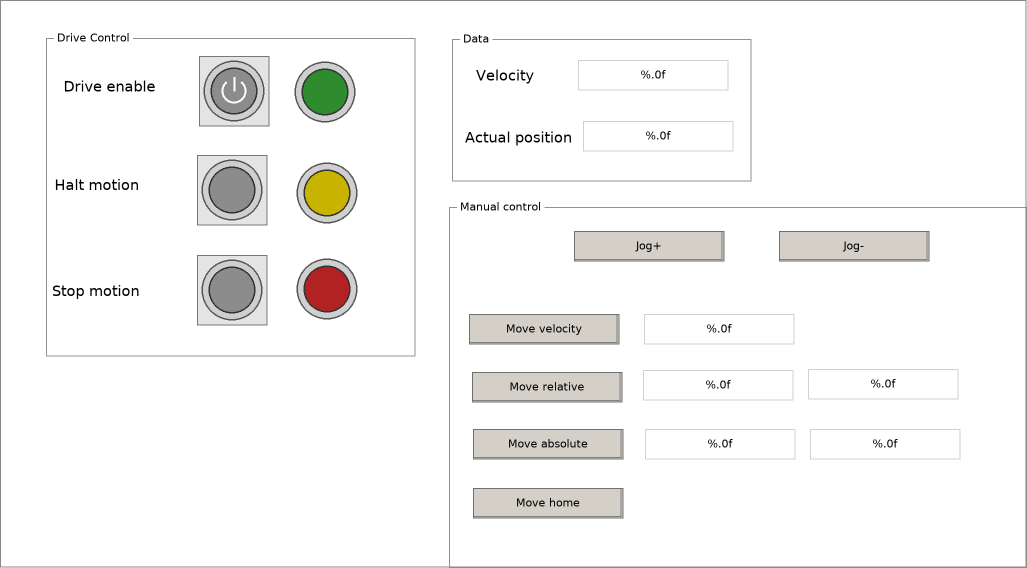
VISUALIZATION HMI  // 1027x568
    GroupBox (46,30 369x326), "Drive Control"
        PowerSwitch (153,26 70x70), variable: MAIN.AxisControl.McPowerEnable, behaviour: TOGGLE, style: Switch-PowerSwitch-Gray
        Lamp1 (244,27 70x70), variable: MAIN.AxisControl.AxisStatus, style: Lamp-Lamp1-Green
        PushSwitch (151,125 70x70), variable: MAIN.AxisControl.ExecuteHalt, behaviour: TOGGLE, style: Switch-PushSwitch-Gray
        PushSwitch (151,225 70x70), variable: MAIN.AxisControl.ExecuteStop, behaviour: TOGGLE, style: Switch-PushSwitch-Gray
        Lamp1 (246,128 70x70), variable: MAIN.AxisControl.McHalt.Done, style: Lamp-Lamp1-Yellow
        Lamp1 (246,224 70x70), variable: MAIN.AxisControl.McStop.Done, style: Lamp-Lamp1-Red
    Label (22,170 150x30), "Halt motion"
    Label (21,276 150x30), "Stop motion"
    Label (44,66 131x41), "Drive enable"
    GroupBox (452,31 299x150), "Data"
        Label (6,32 94x25), "Velocity"
        Textfield (126,29 150x30), "%.0f", text variable: MAIN.AxisControl.ActualVelocity
        Label (11,95 111x23), "Actual position"
        Textfield (131,90 150x30), "%.0f", text variable: MAIN.AxisControl.ActualPosition
    GroupBox (449,199 578x369), "Manual control"
        Button (125,32 150x30), "Jog+"
            OnMouseDown: toggle MAIN.AxisControl.JogForward
        Button (330,32 150x30), "Jog-"
            OnMouseDown: toggle MAIN.AxisControl.JogBackward
        Button (20,115 150x30), "Move velocity"
            OnMouseDown: toggle MAIN.AxisControl.ExecuteVelocity
        Textfield (195,115 150x30), "%.0f", tooltip "Type velocity", text variable: MAIN.AxisControl.Velocity
            OnMouseClick: write the text variable via Edit, min 0, max 50
        Button (23,173 150x30), "Move relative"
            OnMouseDown: toggle MAIN.AxisControl.ExecuteRelative
        Textfield (194,171 150x30), "%.0f", tooltip "Type relative pos", text variable: MAIN.AxisControl.RelativeDistance
            OnMouseClick: write the text variable via Edit
        Button (24,230 150x30), "Move absolute"
            OnMouseDown: toggle MAIN.AxisControl.ExecuteAbsolute
        Textfield (196,230 150x30), "%.0f", tooltip "Type absolute pos", text variable: MAIN.AxisControl.AbsolutePosition
            OnMouseClick: write the text variable via Edit
        Button (24,289 150x30), "Move home"
            OnMouseDown: toggle MAIN.AxisControl.ExecuteHome
        Textfield (359,170 150x30), "%.0f", tooltip "Type relative velocity", text variable: MAIN.AxisControl.RelativeVelocity
            OnMouseClick: write the text variable via Edit
        Textfield (361,230 150x30), "%.0f", tooltip "Type absolute velocity", text variable: MAIN.AxisControl.AbsoluteVelocity
            OnMouseClick: write the text variable via Edit
END_VISUALIZATION

(* stored: Version 1.1.0.1, ProductVersion 3.1.4024.13
   Visu HMI: Id {5cfdce4e-1e29-40f5-98cc-0ad19fd4d836} *)
